(* Logix 5000 project; controller Commerford_topping_5477_V3 vendor 1 type 14 code 222 rev 33.11; software revision 33.02; part 4 of 6 *)
(* UN6_EM3_Color_2, continued *)

ROUTINE _EP_Running   (* ladder *)
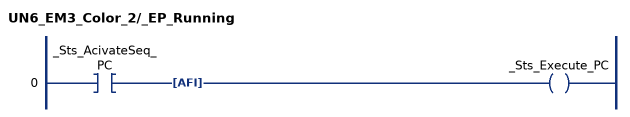
   0: XIC(_Sts_AcivateSeq_PC)AFI()OTE(_Sts_Execute_PC);
END_ROUTINE

ROUTINE _FaultHandler   (* ladder *)
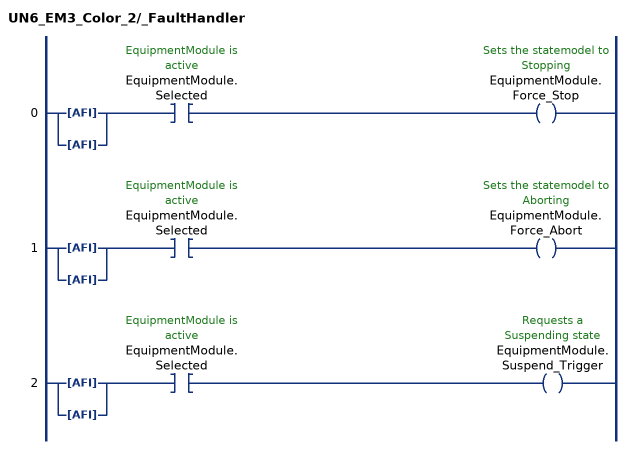
   0: [AFI() ,AFI() ]XIC(EquipmentModule.Selected)OTE(EquipmentModule.Force_Stop);
   1: [AFI() ,AFI() ]XIC(EquipmentModule.Selected)OTE(EquipmentModule.Force_Abort);
   2: [AFI() ,AFI() ]XIC(EquipmentModule.Selected)OTE(EquipmentModule.Suspend_Trigger);
END_ROUTINE

ROUTINE _INOUT   (* ladder *)
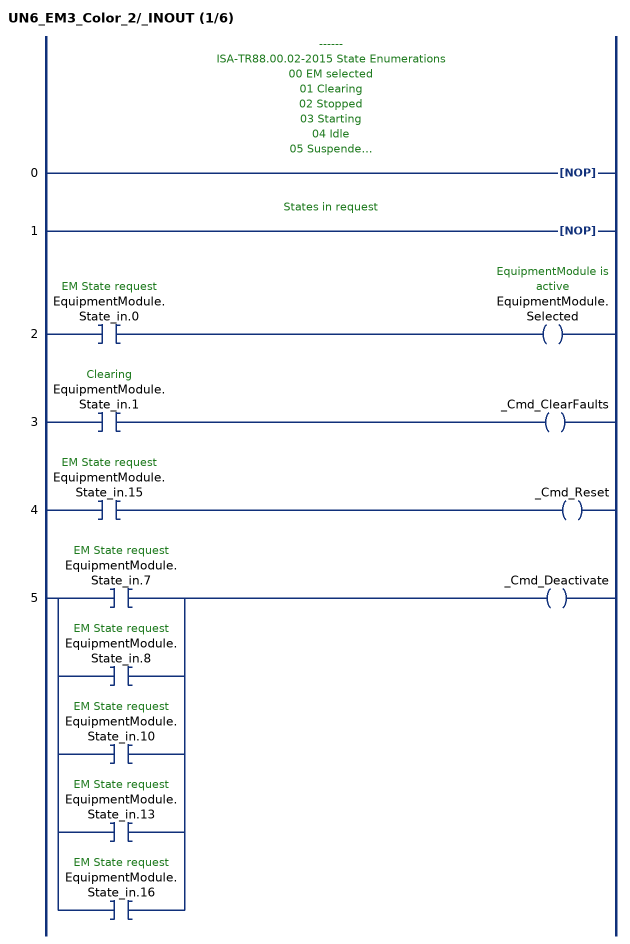
   // ------
   // ISA-TR88.00.02-2015 State Enumerations
   // 00 EM selected
   // 01 Clearing
   // 02 Stopped
   // 03 Starting
   // 04 Idle
   // 05 Suspended
   // 06 Execute
   // 07 Stopping
   // 08 Aborting
   // 09 Aborted
   // 10 Holding
   // 11 Held
   // 12 UnHolding
   // 13 Suspending
   // 14 Unsuspending
   // 15 Resetting
   // 16 Completing
   // 17 Complete
   // 18 Undefined
   // 19 Undefined
   // 20 Suspend trigger
   // 21 Faulted
   // 22 Force stop
   // 23 Force abort
   // 24 Reset signal
   // 31 Undefined
   // ------
   0: NOP();
   // States in request
   1: NOP();
   2: XIC(EquipmentModule.State_in.0)OTE(EquipmentModule.Selected);
   3: XIC(EquipmentModule.State_in.1)OTE(_Cmd_ClearFaults);
   4: XIC(EquipmentModule.State_in.15)OTE(_Cmd_Reset);
   5: [XIC(EquipmentModule.State_in.7) ,XIC(EquipmentModule.State_in.8) ,XIC(EquipmentModule.State_in.10) ,XIC(EquipmentModule.State_in.13) ,XIC(EquipmentModule.State_in.16) ]OTE(_Cmd_Deactivate);
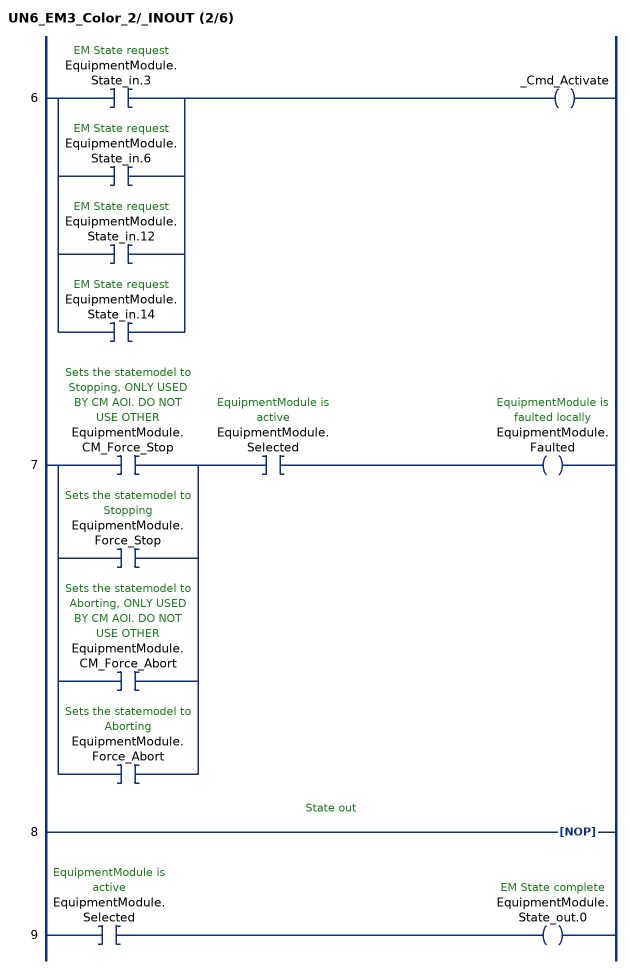
   6: [XIC(EquipmentModule.State_in.3) ,XIC(EquipmentModule.State_in.6) ,XIC(EquipmentModule.State_in.12) ,XIC(EquipmentModule.State_in.14) ]OTE(_Cmd_Activate);
   7: [XIC(EquipmentModule.CM_Force_Stop) ,XIC(EquipmentModule.Force_Stop) ,XIC(EquipmentModule.CM_Force_Abort) ,XIC(EquipmentModule.Force_Abort) ]XIC(EquipmentModule.Selected)OTE(EquipmentModule.Faulted);
   // State out
   8: NOP();
   9: XIC(EquipmentModule.Selected)OTE(EquipmentModule.State_out.0);
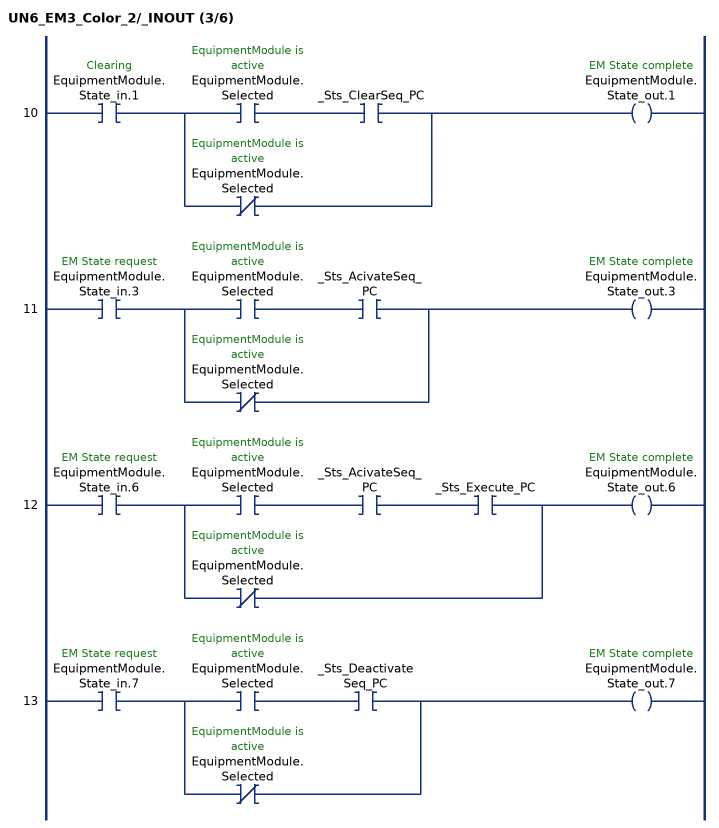
   10: XIC(EquipmentModule.State_in.1)[XIC(EquipmentModule.Selected) XIC(_Sts_ClearSeq_PC) ,XIO(EquipmentModule.Selected) ]OTE(EquipmentModule.State_out.1);
   11: XIC(EquipmentModule.State_in.3)[XIC(EquipmentModule.Selected) XIC(_Sts_AcivateSeq_PC) ,XIO(EquipmentModule.Selected) ]OTE(EquipmentModule.State_out.3);
   12: XIC(EquipmentModule.State_in.6)[XIC(EquipmentModule.Selected) XIC(_Sts_AcivateSeq_PC) XIC(_Sts_Execute_PC) ,XIO(EquipmentModule.Selected) ]OTE(EquipmentModule.State_out.6);
   13: XIC(EquipmentModule.State_in.7)[XIC(EquipmentModule.Selected) XIC(_Sts_DeactivateSeq_PC) ,XIO(EquipmentModule.Selected) ]OTE(EquipmentModule.State_out.7);
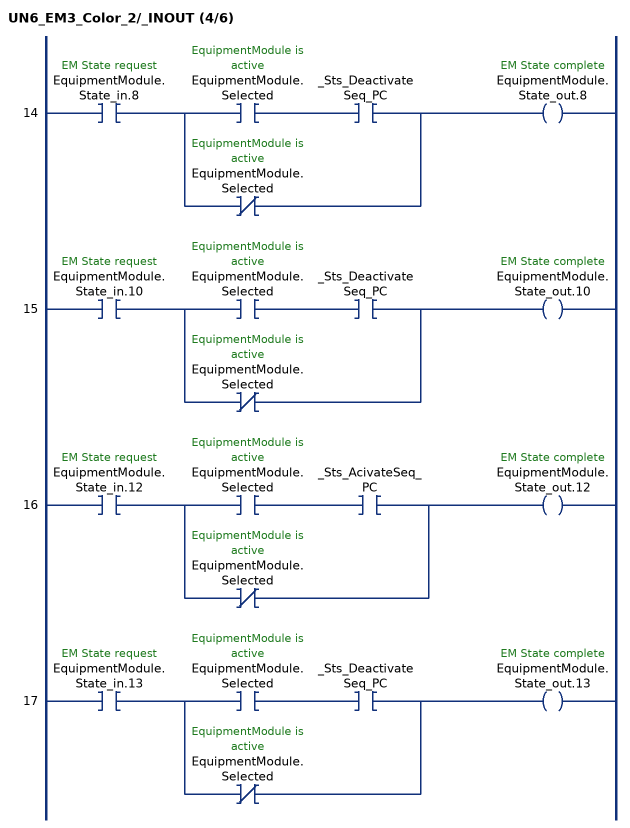
   14: XIC(EquipmentModule.State_in.8)[XIC(EquipmentModule.Selected) XIC(_Sts_DeactivateSeq_PC) ,XIO(EquipmentModule.Selected) ]OTE(EquipmentModule.State_out.8);
   15: XIC(EquipmentModule.State_in.10)[XIC(EquipmentModule.Selected) XIC(_Sts_DeactivateSeq_PC) ,XIO(EquipmentModule.Selected) ]OTE(EquipmentModule.State_out.10);
   16: XIC(EquipmentModule.State_in.12)[XIC(EquipmentModule.Selected) XIC(_Sts_AcivateSeq_PC) ,XIO(EquipmentModule.Selected) ]OTE(EquipmentModule.State_out.12);
   17: XIC(EquipmentModule.State_in.13)[XIC(EquipmentModule.Selected) XIC(_Sts_DeactivateSeq_PC) ,XIO(EquipmentModule.Selected) ]OTE(EquipmentModule.State_out.13);
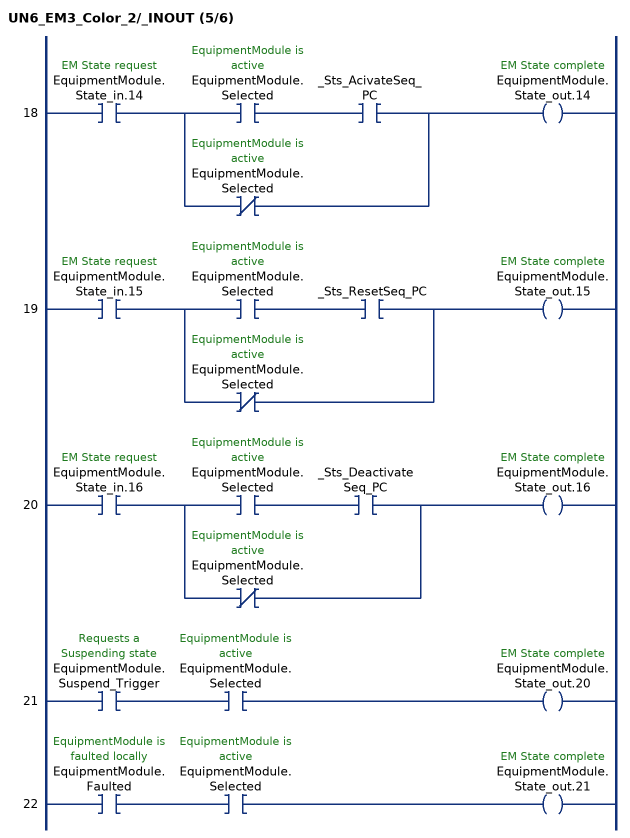
   18: XIC(EquipmentModule.State_in.14)[XIC(EquipmentModule.Selected) XIC(_Sts_AcivateSeq_PC) ,XIO(EquipmentModule.Selected) ]OTE(EquipmentModule.State_out.14);
   19: XIC(EquipmentModule.State_in.15)[XIC(EquipmentModule.Selected) XIC(_Sts_ResetSeq_PC) ,XIO(EquipmentModule.Selected) ]OTE(EquipmentModule.State_out.15);
   20: XIC(EquipmentModule.State_in.16)[XIC(EquipmentModule.Selected) XIC(_Sts_DeactivateSeq_PC) ,XIO(EquipmentModule.Selected) ]OTE(EquipmentModule.State_out.16);
   21: XIC(EquipmentModule.Suspend_Trigger)XIC(EquipmentModule.Selected)OTE(EquipmentModule.State_out.20);
   22: XIC(EquipmentModule.Faulted)XIC(EquipmentModule.Selected)OTE(EquipmentModule.State_out.21);
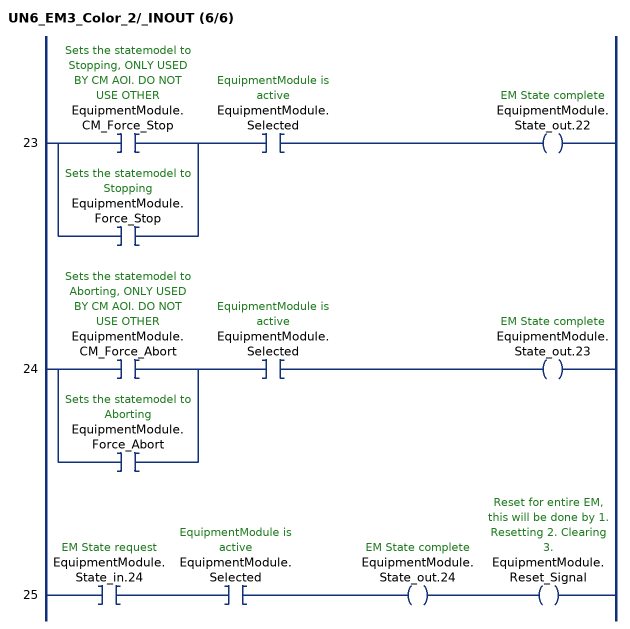
   23: [XIC(EquipmentModule.CM_Force_Stop) ,XIC(EquipmentModule.Force_Stop) ]XIC(EquipmentModule.Selected)OTE(EquipmentModule.State_out.22);
   24: [XIC(EquipmentModule.CM_Force_Abort) ,XIC(EquipmentModule.Force_Abort) ]XIC(EquipmentModule.Selected)OTE(EquipmentModule.State_out.23);
   25: XIC(EquipmentModule.State_in.24)XIC(EquipmentModule.Selected)OTE(EquipmentModule.State_out.24)OTE(EquipmentModule.Reset_Signal);
END_ROUTINE

ROUTINE Main   (* ladder *)
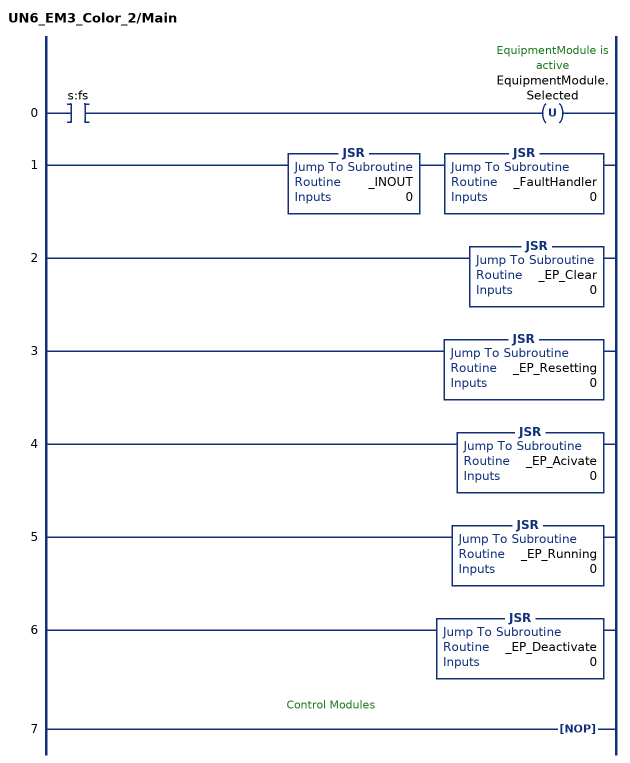
   0: XIC(s:fs)OTU(EquipmentModule.Selected);
   1: JSR(_INOUT,0)JSR(_FaultHandler,0);
   2: JSR(_EP_Clear,0);
   3: JSR(_EP_Resetting,0);
   4: JSR(_EP_Acivate,0);
   5: JSR(_EP_Running,0);
   6: JSR(_EP_Deactivate,0);
   // Control Modules
   7: NOP();
END_ROUTINE
END_PROGRAM

PROGRAM UN6_EM4_Color_3   (* main routine Main *)
// Color_3, generated by G.E.M
VAR
   _Cmd_Activate : BOOL;
   _Cmd_ClearFaults : BOOL;
   _Cmd_Deactivate : BOOL;
   _Cmd_Reset : BOOL;
   _Sts_AcivateSeq_PC : BOOL;
   _Sts_ClearSeq_PC : BOOL;
   _Sts_DeactivateSeq_PC : BOOL;
   _Sts_Execute_PC : BOOL;
   _Sts_ResetSeq_PC : BOOL;
END_VAR
VAR {public}
   EquipmentModule : EquipmentModule := (Selected := 1, State_in := 2#0000_0000_0000_0000_0000_0000_0000_0101, State_out := 2#0000_0000_0000_0000_0000_0000_0000_0001, _SEQ.Clearing := -1, _SEQ.Activating := -1, _SEQ.Deactivating := -1, _SEQ.Resetting := -1);
        .State_in.1   // Clearing
END_VAR

ROUTINE _EP_Acivate   (* ladder *)
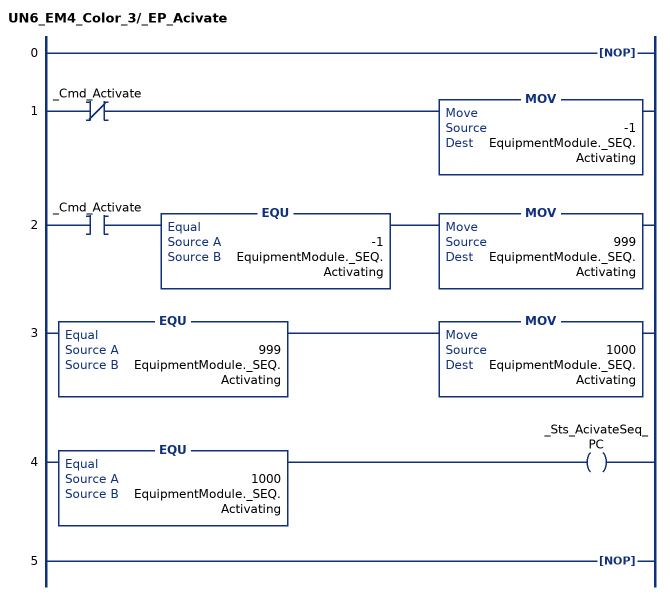
   0: NOP();
   1: XIO(_Cmd_Activate)MOV(-1,EquipmentModule._SEQ.Activating);
   2: XIC(_Cmd_Activate)EQU(-1,EquipmentModule._SEQ.Activating)MOV(999,EquipmentModule._SEQ.Activating);
   3: EQU(999,EquipmentModule._SEQ.Activating)MOV(1000,EquipmentModule._SEQ.Activating);
   4: EQU(1000,EquipmentModule._SEQ.Activating)OTE(_Sts_AcivateSeq_PC);
   5: NOP();
END_ROUTINE

ROUTINE _EP_Clear   (* ladder *)
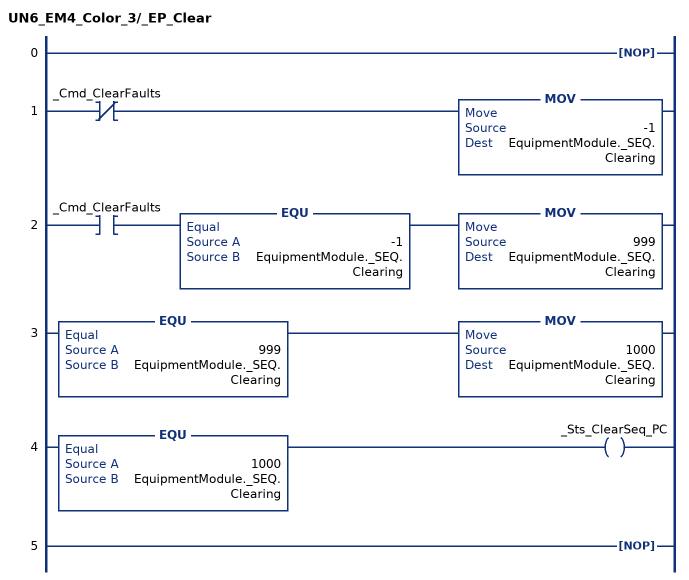
   0: NOP();
   1: XIO(_Cmd_ClearFaults)MOV(-1,EquipmentModule._SEQ.Clearing);
   2: XIC(_Cmd_ClearFaults)EQU(-1,EquipmentModule._SEQ.Clearing)MOV(999,EquipmentModule._SEQ.Clearing);
   3: EQU(999,EquipmentModule._SEQ.Clearing)MOV(1000,EquipmentModule._SEQ.Clearing);
   4: EQU(1000,EquipmentModule._SEQ.Clearing)OTE(_Sts_ClearSeq_PC);
   5: NOP();
END_ROUTINE

ROUTINE _EP_Deactivate   (* ladder *)
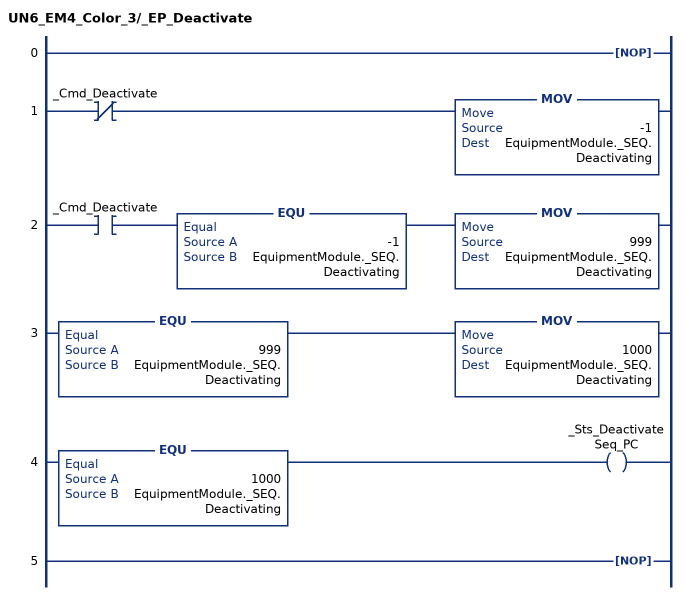
   0: NOP();
   1: XIO(_Cmd_Deactivate)MOV(-1,EquipmentModule._SEQ.Deactivating);
   2: XIC(_Cmd_Deactivate)EQU(-1,EquipmentModule._SEQ.Deactivating)MOV(999,EquipmentModule._SEQ.Deactivating);
   3: EQU(999,EquipmentModule._SEQ.Deactivating)MOV(1000,EquipmentModule._SEQ.Deactivating);
   4: EQU(1000,EquipmentModule._SEQ.Deactivating)OTE(_Sts_DeactivateSeq_PC);
   5: NOP();
END_ROUTINE

ROUTINE _EP_Resetting   (* ladder *)
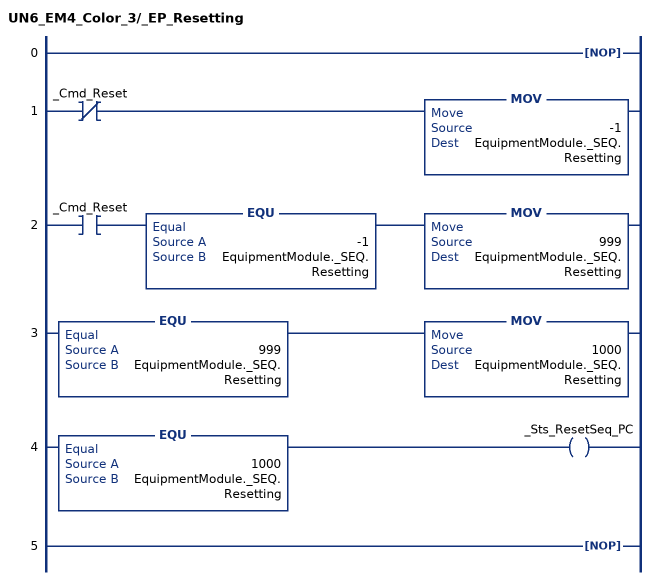
   0: NOP();
   1: XIO(_Cmd_Reset)MOV(-1,EquipmentModule._SEQ.Resetting);
   2: XIC(_Cmd_Reset)EQU(-1,EquipmentModule._SEQ.Resetting)MOV(999,EquipmentModule._SEQ.Resetting);
   3: EQU(999,EquipmentModule._SEQ.Resetting)MOV(1000,EquipmentModule._SEQ.Resetting);
   4: EQU(1000,EquipmentModule._SEQ.Resetting)OTE(_Sts_ResetSeq_PC);
   5: NOP();
END_ROUTINE

ROUTINE _EP_Running   (* ladder *)
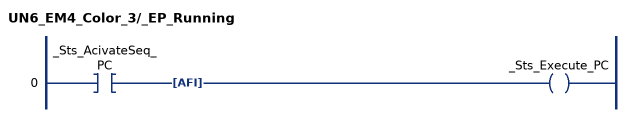
   0: XIC(_Sts_AcivateSeq_PC)AFI()OTE(_Sts_Execute_PC);
END_ROUTINE

ROUTINE _FaultHandler   (* ladder *)
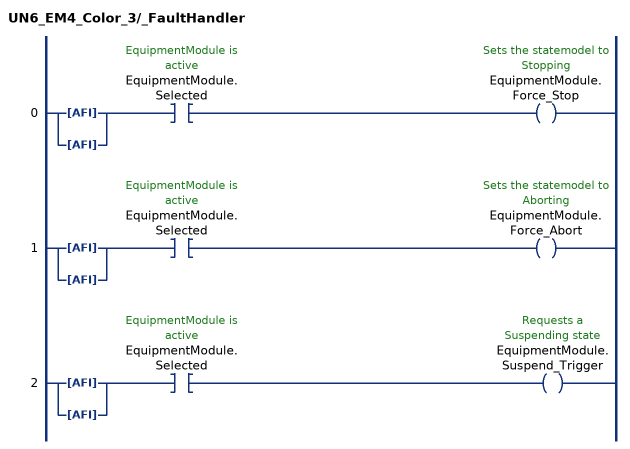
   0: [AFI() ,AFI() ]XIC(EquipmentModule.Selected)OTE(EquipmentModule.Force_Stop);
   1: [AFI() ,AFI() ]XIC(EquipmentModule.Selected)OTE(EquipmentModule.Force_Abort);
   2: [AFI() ,AFI() ]XIC(EquipmentModule.Selected)OTE(EquipmentModule.Suspend_Trigger);
END_ROUTINE

ROUTINE _INOUT   (* ladder *)
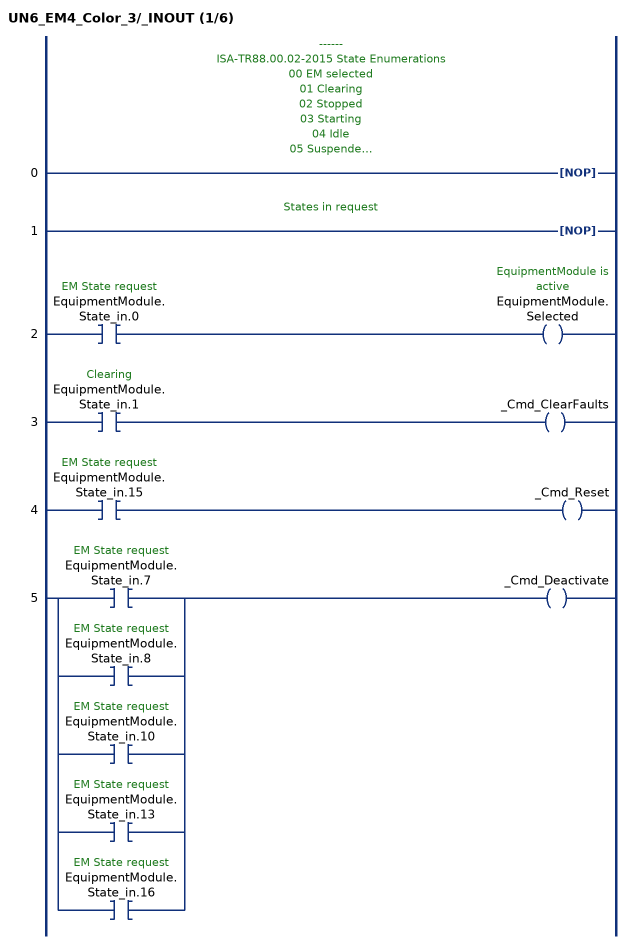
   // ------
   // ISA-TR88.00.02-2015 State Enumerations
   // 00 EM selected
   // 01 Clearing
   // 02 Stopped
   // 03 Starting
   // 04 Idle
   // 05 Suspended
   // 06 Execute
   // 07 Stopping
   // 08 Aborting
   // 09 Aborted
   // 10 Holding
   // 11 Held
   // 12 UnHolding
   // 13 Suspending
   // 14 Unsuspending
   // 15 Resetting
   // 16 Completing
   // 17 Complete
   // 18 Undefined
   // 19 Undefined
   // 20 Suspend trigger
   // 21 Faulted
   // 22 Force stop
   // 23 Force abort
   // 24 Reset signal
   // 31 Undefined
   // ------
   0: NOP();
   // States in request
   1: NOP();
   2: XIC(EquipmentModule.State_in.0)OTE(EquipmentModule.Selected);
   3: XIC(EquipmentModule.State_in.1)OTE(_Cmd_ClearFaults);
   4: XIC(EquipmentModule.State_in.15)OTE(_Cmd_Reset);
   5: [XIC(EquipmentModule.State_in.7) ,XIC(EquipmentModule.State_in.8) ,XIC(EquipmentModule.State_in.10) ,XIC(EquipmentModule.State_in.13) ,XIC(EquipmentModule.State_in.16) ]OTE(_Cmd_Deactivate);
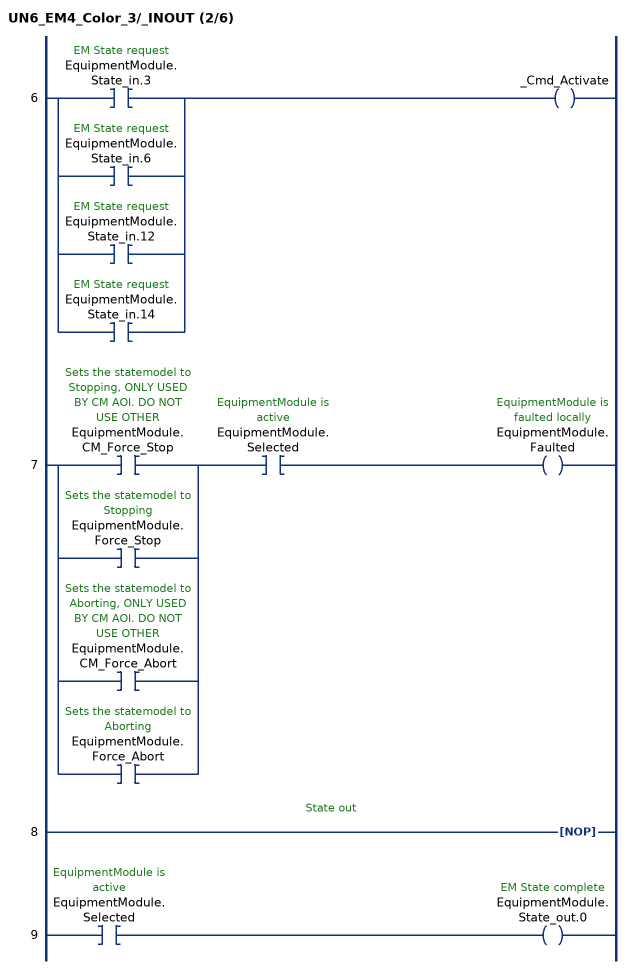
   6: [XIC(EquipmentModule.State_in.3) ,XIC(EquipmentModule.State_in.6) ,XIC(EquipmentModule.State_in.12) ,XIC(EquipmentModule.State_in.14) ]OTE(_Cmd_Activate);
   7: [XIC(EquipmentModule.CM_Force_Stop) ,XIC(EquipmentModule.Force_Stop) ,XIC(EquipmentModule.CM_Force_Abort) ,XIC(EquipmentModule.Force_Abort) ]XIC(EquipmentModule.Selected)OTE(EquipmentModule.Faulted);
   // State out
   8: NOP();
   9: XIC(EquipmentModule.Selected)OTE(EquipmentModule.State_out.0);
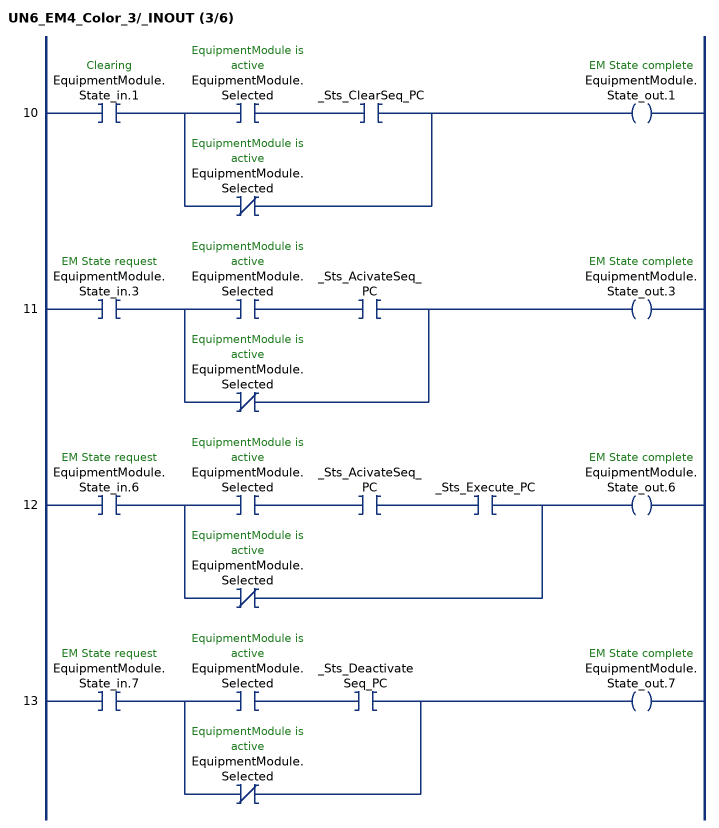
   10: XIC(EquipmentModule.State_in.1)[XIC(EquipmentModule.Selected) XIC(_Sts_ClearSeq_PC) ,XIO(EquipmentModule.Selected) ]OTE(EquipmentModule.State_out.1);
   11: XIC(EquipmentModule.State_in.3)[XIC(EquipmentModule.Selected) XIC(_Sts_AcivateSeq_PC) ,XIO(EquipmentModule.Selected) ]OTE(EquipmentModule.State_out.3);
   12: XIC(EquipmentModule.State_in.6)[XIC(EquipmentModule.Selected) XIC(_Sts_AcivateSeq_PC) XIC(_Sts_Execute_PC) ,XIO(EquipmentModule.Selected) ]OTE(EquipmentModule.State_out.6);
   13: XIC(EquipmentModule.State_in.7)[XIC(EquipmentModule.Selected) XIC(_Sts_DeactivateSeq_PC) ,XIO(EquipmentModule.Selected) ]OTE(EquipmentModule.State_out.7);
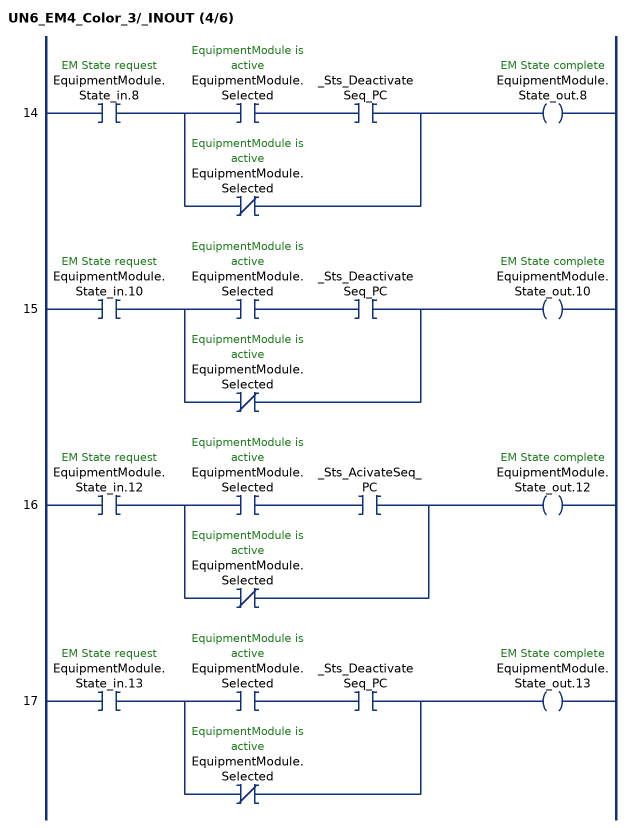
   14: XIC(EquipmentModule.State_in.8)[XIC(EquipmentModule.Selected) XIC(_Sts_DeactivateSeq_PC) ,XIO(EquipmentModule.Selected) ]OTE(EquipmentModule.State_out.8);
   15: XIC(EquipmentModule.State_in.10)[XIC(EquipmentModule.Selected) XIC(_Sts_DeactivateSeq_PC) ,XIO(EquipmentModule.Selected) ]OTE(EquipmentModule.State_out.10);
   16: XIC(EquipmentModule.State_in.12)[XIC(EquipmentModule.Selected) XIC(_Sts_AcivateSeq_PC) ,XIO(EquipmentModule.Selected) ]OTE(EquipmentModule.State_out.12);
   17: XIC(EquipmentModule.State_in.13)[XIC(EquipmentModule.Selected) XIC(_Sts_DeactivateSeq_PC) ,XIO(EquipmentModule.Selected) ]OTE(EquipmentModule.State_out.13);
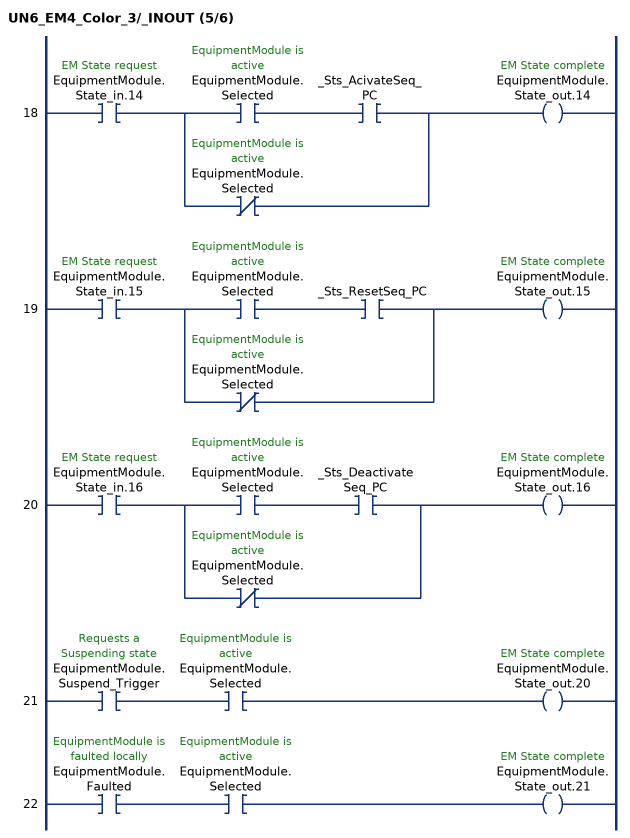
   18: XIC(EquipmentModule.State_in.14)[XIC(EquipmentModule.Selected) XIC(_Sts_AcivateSeq_PC) ,XIO(EquipmentModule.Selected) ]OTE(EquipmentModule.State_out.14);
   19: XIC(EquipmentModule.State_in.15)[XIC(EquipmentModule.Selected) XIC(_Sts_ResetSeq_PC) ,XIO(EquipmentModule.Selected) ]OTE(EquipmentModule.State_out.15);
   20: XIC(EquipmentModule.State_in.16)[XIC(EquipmentModule.Selected) XIC(_Sts_DeactivateSeq_PC) ,XIO(EquipmentModule.Selected) ]OTE(EquipmentModule.State_out.16);
   21: XIC(EquipmentModule.Suspend_Trigger)XIC(EquipmentModule.Selected)OTE(EquipmentModule.State_out.20);
   22: XIC(EquipmentModule.Faulted)XIC(EquipmentModule.Selected)OTE(EquipmentModule.State_out.21);
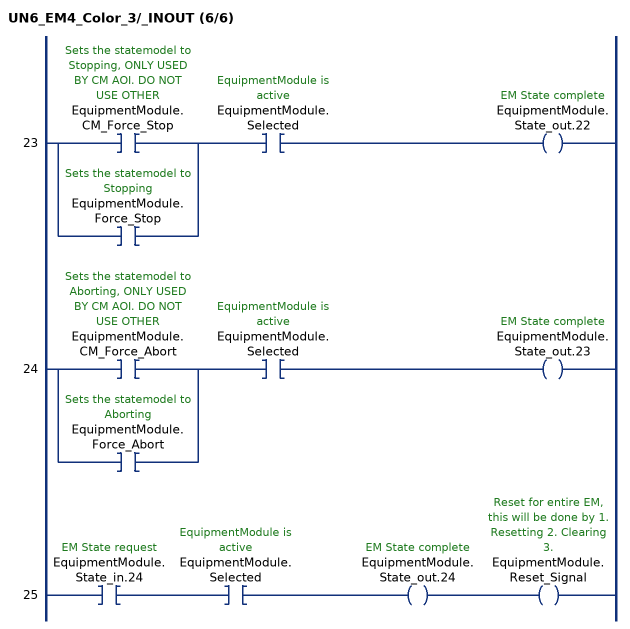
   23: [XIC(EquipmentModule.CM_Force_Stop) ,XIC(EquipmentModule.Force_Stop) ]XIC(EquipmentModule.Selected)OTE(EquipmentModule.State_out.22);
   24: [XIC(EquipmentModule.CM_Force_Abort) ,XIC(EquipmentModule.Force_Abort) ]XIC(EquipmentModule.Selected)OTE(EquipmentModule.State_out.23);
   25: XIC(EquipmentModule.State_in.24)XIC(EquipmentModule.Selected)OTE(EquipmentModule.State_out.24)OTE(EquipmentModule.Reset_Signal);
END_ROUTINE
